(* IEC 61131-3 sources: programs/VI-54/VI-54_20171205/VI-54_20171205/Stations/Screen/LseClass170718/Class/SaveAcces, 1 file *)

(* ---- SaveAcces.st ---- *)
(*!
<Class
	Name               = "SaveAcces"
	Revision           = "2.1"
	RealtimeTask       = "false"
	CyclicTask         = "false"
	BackgroundTask     = "true"
	DefBackground      = "100 ms"
	Sigmatek           = "false"
	OSInterface        = "false"
	HighPriority       = "false"
	Automatic          = "false"
	UpdateMode         = "Prescan"
	SharedCommandTable = "true"
	Objectsize         = "(550,120)">
	<Channels>
		<Server Name="CodeOk" Visualized="true" Initialize="false" WriteProtected="true" Retentive="false"/>
		<Server Name="CopyNbr" Visualized="true" Initialize="false" WriteProtected="false" Retentive="false"/>
		<Server Name="SaveCmd" Visualized="true" Initialize="false" WriteProtected="false" Retentive="false"/>
		<Server Name="SaveCode" Visualized="true" Initialize="false" WriteProtected="false" Retentive="false"/>
		<Client Name="Comm_RecipeHandle" Required="true" Internal="false"/>
		<Client Name="vDelActRecept" Required="false" Internal="false"/>
		<Client Name="vLevel" Required="false" Internal="false"/>
		<Client Name="vSaveReceptNr" Required="true" Internal="false"/>
	</Channels>
</Class>
*)
SaveAcces : CLASS
  //Servers:
	SaveCode 	: SvrChCmd_DINT;
	SaveCmd 	: SvrCh_DINT;
	CopyNbr 	: SvrCh_DINT;
	CodeOk 	: SvrCh_DINT;
  //Clients:
	Comm_RecipeHandle 	: CltChCmd_RecipeHandle;
	vSaveReceptNr 	: CltCh_DINT;
	vDelActRecept 	: CltCh_DINT;
	vLevel 	: CltCh_DINT;
  //Variables:
		WriteValue 	: DINT;
		FileOSState 	: DINT;
		ActRecipeNbr 	: DINT;
		OldLoadProg 	: DINT;
  //Functions:

	FUNCTION VIRTUAL GLOBAL Init;

	FUNCTION VIRTUAL GLOBAL Background
		VAR_INPUT
			EAX 	: UDINT;
		END_VAR
		VAR_OUTPUT
			state (EAX) 	: UDINT;
		END_VAR;

	FUNCTION VIRTUAL GLOBAL SaveCmd::Write
		VAR_INPUT
			input (EAX) 	: DINT;
		END_VAR
		VAR_OUTPUT
			result (EAX) 	: DINT;
		END_VAR;
  //Tables:
	FUNCTION @STD
		VAR_OUTPUT
			ret_code	: CONFSTATES;
		END_VAR;
	FUNCTION GLOBAL TAB @CT_;
END_CLASS;

#pragma usingLtd RecipeHandle

FUNCTION VIRTUAL GLOBAL SaveAcces::Init

  SaveCmd := -1;

END_FUNCTION

FUNCTION VIRTUAL GLOBAL SaveAcces::SaveCmd::Write
	VAR_INPUT
		input (EAX) 	: DINT;
	END_VAR
	VAR_OUTPUT
		result (EAX) 	: DINT;
	END_VAR

	SaveCmd := input;

  ActRecipeNbr := Comm_RecipeHandle.ReadActRecipe();

  case SaveCmd of
  00:// no action

  01:// save actuele recipe
    if CodeOk = 1 then
      vSaveReceptNr := ActRecipeNbr;
      vSaveReceptNr.write( vSaveReceptNr);
    end_if;

  02: // Copy actual recipe to new recipe nbr
    if CodeOk = 1 then
      vSaveReceptNr := CopyNbr;
      vSaveReceptNr.write( CopyNbr);
    end_if;

  03: // Delete recipe
    if CodeOk = 1 then
      vDelActRecept := ActRecipeNbr;
      vDelActRecept.Write(input:= vDelActRecept);
    end_if;

  04:// save actuele recipe
    vSaveReceptNr := ActRecipeNbr;
    vSaveReceptNr.write( vSaveReceptNr);

  end_case;

  SaveCmd := -1;
  SaveCode := 0;

 	result := SaveCmd;

END_FUNCTION

FUNCTION VIRTUAL GLOBAL SaveAcces::Background
	VAR_INPUT
		EAX 	: UDINT;
	END_VAR
	VAR_OUTPUT
		state (EAX) 	: UDINT;
	END_VAR

  // check code..
  if IsClientConnected(#vLevel ) then
    vLevel := vLevel.Read();
  end_if;

  // bij juiste level is saven ook mogelijk
  if vLevel >= OPPERATOR then
    CodeOk := 1;
  elsif SaveCode = _SaveCode then
    CodeOk := 1;
  else
    CodeOk := 0;
  end_if;

  // When program is changed, change also CopyNbr
  if Comm_RecipeHandle.LoadProgNbr <> OldLoadProg then
    CopyNbr := Comm_RecipeHandle.LoadProgNbr;
    OldLoadProg := Comm_RecipeHandle.LoadProgNbr;
  end_if;

	state := READY;

END_FUNCTION
